FUNCTION F_Add : INT
VAR_INPUT
	nFirstNum : INT;
	nSecondNum : INT;
END_VAR
VAR_OUTPUT
	nResult : INT;
END_VAR
VAR
END_VAR

nResult := nFirstNum + nSecondNum;

END_FUNCTION

(* stored: Version 1.1.0.1, ProductVersion 3.1.4024.16
   POU F_Add: Id {6051fc38-ff1c-466b-8fb6-384cb470a531}, SpecialFunc None *)
